// Mitsubishi GX Works2 project: BookEX6_8 Function   PLC: Q13UDV

// global labels: Global
VAR_GLOBAL
  bVar0 AT M5000 : BOOL;
  abArray0 AT M5010 : ARRAY [0..49] OF BOOL;
  sStr0 AT D5000 : STRING[199];
  sStr1 AT D5100 : STRING[199];
  sStr2 AT D5200 : STRING[199];
  sStr3 AT D5300 : STRING[199];
  sStr4 AT D5400 : STRING[199];
  sStr5 AT D5500 : STRING[199];
  sStr6 AT D5600 : STRING[199];
  sStr7 AT D5700 : STRING[199];
  sStr8 AT D5800 : STRING[199];
  sStr9 AT D5900 : STRING[199];
  iVar0 AT D4500 : INT;
  iVar1 AT D4501 : INT;
  iVar2 AT D4502 : INT;
  iVar3 AT D4503 : INT;
  iVar4 AT D4504 : INT;
  iVar5 AT D4505 : INT;
  iVar6 AT D4506 : INT;
  iVar7 AT D4507 : INT;
  iVar8 AT D4508 : INT;
  iVar9 AT D4509 : INT;
  dVar0 AT D4510 : DINT;
  dVar1 AT D4512 : DINT;
  dVar2 AT D4514 : DINT;
  dVar3 AT D4516 : DINT;
  dVar4 AT D4518 : DINT;
  dVar5 AT D4520 : DINT;
  dVar6 AT D4522 : DINT;
  dVar7 AT D4524 : DINT;
  dVar8 AT D4526 : DINT;
  dVar9 AT D4528 : DINT;
  wVar0 AT D4530 : WORD;
  wVar1 AT D4531 : WORD;
  wVar2 AT D4532 : WORD;
  wVar3 AT D4533 : WORD;
  wVar4 AT D4534 : WORD;
  wVar5 AT D4535 : WORD;
  wVar6 AT D4536 : WORD;
  wVar7 AT D4537 : WORD;
  wVar8 AT D4538 : WORD;
  wVar9 AT D4539 : WORD;
  dwVar0 AT D4540 : DWORD;
  dwVar1 AT D4542 : DWORD;
  dwVar2 AT D4544 : DWORD;
  dwVar3 AT D4546 : DWORD;
  dwVar4 AT D4548 : DWORD;
  dwVar5 AT D4550 : DWORD;
  dwVar6 AT D4552 : DWORD;
  dwVar7 AT D4554 : DWORD;
  dwVar8 AT D4556 : DWORD;
  dwVar9 AT D4558 : DWORD;
  fsVar0 AT D4560 : REAL;
  fsVar1 AT D4562 : REAL;
  fsVar2 AT D4564 : REAL;
  fsVar3 AT D4566 : REAL;
  fsVar4 AT D4568 : REAL;
  fsVar5 AT D4570 : REAL;
  fsVar6 AT D4572 : REAL;
  fsVar7 AT D4574 : REAL;
  fsVar8 AT D4576 : REAL;
  fsVar9 AT D4578 : REAL;
  fdVar0 AT D4580 : LREAL;
  tTime0 AT D4620 : TIME;
  tTime1 AT D4622 : TIME;
  tTime2 AT D4624 : TIME;
  tTime3 AT D4626 : TIME;
  tTime4 AT D4628 : TIME;
  tTime5 AT D4630 : TIME;
  tTime6 AT D4632 : TIME;
  tTime7 AT D4634 : TIME;
  tTime8 AT D4636 : TIME;
  tTime9 AT D4638 : TIME;
  tTime10 AT D4640 : TIME;
  bVar1 AT M5001 : BOOL;
  bVar2 AT M5002 : BOOL;
  bVar3 AT M5003 : BOOL;
  bVar4 AT M5004 : BOOL;
  bVar5 AT M5005 : BOOL;
  bVar6 AT M5006 : BOOL;
  bVar7 AT M5007 : BOOL;
  bVar8 AT M5008 : BOOL;
  bVar9 AT M5009 : BOOL;
  abArray1 AT M5060 : ARRAY [0..49] OF BOOL;
  abArray2 AT M5110 : ARRAY [0..49] OF BOOL;
  abArray3 AT M5160 : ARRAY [0..49] OF BOOL;
  abArray4 AT M5210 : ARRAY [0..49] OF BOOL;
  abArray5 AT M5260 : ARRAY [0..49] OF BOOL;
  abArray6 AT M5310 : ARRAY [0..49] OF BOOL;
  abArray7 AT M5360 : ARRAY [0..49] OF BOOL;
  abArray8 AT M5410 : ARRAY [0..49] OF BOOL;
  abArray9 AT M5460 : ARRAY [0..49] OF BOOL;
  fdVar1 AT D4584 : LREAL;
  fdVar2 AT D4588 : LREAL;
  fdVar3 AT D4592 : LREAL;
  fdVar4 AT D4596 : LREAL;
  fdVar5 AT D4600 : LREAL;
  fdVar6 AT D4604 : LREAL;
  fdVar7 AT D4608 : LREAL;
  fdVar8 AT D4612 : LREAL;
  fdVar9 AT D4616 : LREAL;
  afsPen0 AT D2000 : ARRAY [0..499] OF REAL;
  afsPen1 AT D3000 : ARRAY [0..499] OF REAL;
END_VAR
// user libraries (not included): HMI

FUNCTION ACOSH
VAR_INPUT
  fs_IN : REAL;
END_VAR
VAR
  fsTemp1 : REAL;
  fsTemp2 : REAL;
END_VAR
;(* ACOSH *)
ACOSH := LN(fs_IN + SQRT(fs_IN * fs_IN - 1.0));
END_FUNCTION

FUNCTION ASINH
VAR_INPUT
  fs_IN : REAL;
END_VAR
VAR
  fsTemp1 : REAL;
  fsTemp2 : REAL;
END_VAR
;(* ASINH *)
ASINH := LN(fs_IN + SQRT(fs_IN * fs_IN + 1.0));
END_FUNCTION

FUNCTION ATANH
VAR_INPUT
  fs_IN : REAL;
END_VAR
VAR
  fsTemp1 : REAL;
  fsTemp2 : REAL;
END_VAR
;(* ATANH *)
ATANH := LN((1.0 + fs_IN)/(1.0 - fs_IN)) / 2.0;
END_FUNCTION

FUNCTION COSH
VAR_INPUT
  fs_IN : REAL;
END_VAR
VAR
  fsTemp1 : REAL;
  fsTemp2 : REAL;
END_VAR
;(* COSH *)
EXP_E(TRUE, fs_IN, fsTemp1); 
COSH := (1.0 / fsTemp1+fsTemp1) / 2.0;
END_FUNCTION

FUNCTION Day2Time
VAR_INPUT
  fs_IN : REAL;
END_VAR
;
Day2Time := DINT_TO_TIME(REAL_TO_DINT(fs_IN * 86400000.0));
END_FUNCTION

FUNCTION EXP10
VAR_INPUT
  fs_IN : REAL;
END_VAR
VAR
  fsTemp : REAL;
END_VAR
;
EXP_E(TRUE, fs_IN * 2.302585, fsTemp);
EXP10 := fsTemp;
END_FUNCTION

FUNCTION Overlap
VAR_INPUT
  CPos1 : INT;
  CPos2 : INT;
  TPos1 : INT;
  TPos2 : INT;
END_VAR
VAR
  tsPos : INT;
  tePos : INT;
END_VAR
VAR_INPUT
  Safe : INT;
END_VAR
VAR
  tst1 : BOOL;
  tst2 : BOOL;
  tst3 : BOOL;
  tst4 : BOOL;
  csPos : INT;
  cePos : INT;
END_VAR
;
IF TPos1 < TPos2 THEN
	tsPos := TPos1;
	tePos := TPos2;
ELSE
	tsPos := TPos2;
	tePos := TPos1;
END_IF;
IF CPos1 < CPos2 THEN
	csPos := CPos1;
	cePos := CPos2;
ELSE
	csPos := CPos2;
	cePos := CPos1;
END_IF;

tst1 := csPos >= tsPos AND csPos <= tePos;
tst2 := cePos >= tsPos AND cePos <= tePos;
tst3 := ABS(tsPos - cePos) <= Safe;
tst4 := ABS(tePos - csPos) <= Safe;

IF tst1 OR tst2 OR tst3 OR tst4 THEN
	Overlap := TRUE;
ELSE
	Overlap := FALSE;
END_IF;
END_FUNCTION

FUNCTION SINH
VAR_INPUT
  fs_IN : REAL;
END_VAR
VAR
  fsTemp1 : REAL;
  fsTemp2 : REAL;
END_VAR
;(* SINH *)
IF ABS(fs_IN) < 0.002 THEN
	SINH := fs_IN;
ELSE
	EXP_E(TRUE, fs_IN, fsTemp1); 
	EXP_E(TRUE, -fs_IN, fsTemp2); 
	SINH := (fsTemp1 - fsTemp2) / 2.0;
END_IF;
END_FUNCTION

FUNCTION SqrtN
VAR_INPUT
  fs_IN : REAL;
  i_IN : INT;
END_VAR
VAR
  fsTemp : REAL;
END_VAR
;
IF i_IN > 0 THEN
	fsTemp := 1.0 / INT_TO_REAL(i_IN);
	SqrtN := EXPT(fs_IN, fsTemp);
ELSE
	SqrtN := 0.0;
END_IF;
END_FUNCTION

FUNCTION TANH
VAR_INPUT
  fs_IN : REAL;
END_VAR
VAR
  fsTemp1 : REAL;
  fsTemp2 : REAL;
END_VAR
;(* TANH *)
IF fs_IN > 20.0 THEN
	TANH := 1.0;
ELSIF fs_IN < -20.0 THEN
	TANH := -1.0;
ELSE
	EXP_E(TRUE, fs_IN * 2.0, fsTemp1); 
	TANH := 1.0 - 2.0 / (fsTemp1 + 1.0);
END_IF;
END_FUNCTION

PROGRAM ExABS
(* structured ladder/FBD written out as ST: instructions are called as NAME(EN, inputs, outputs); _pN, _eN, _tN stand for wires *)
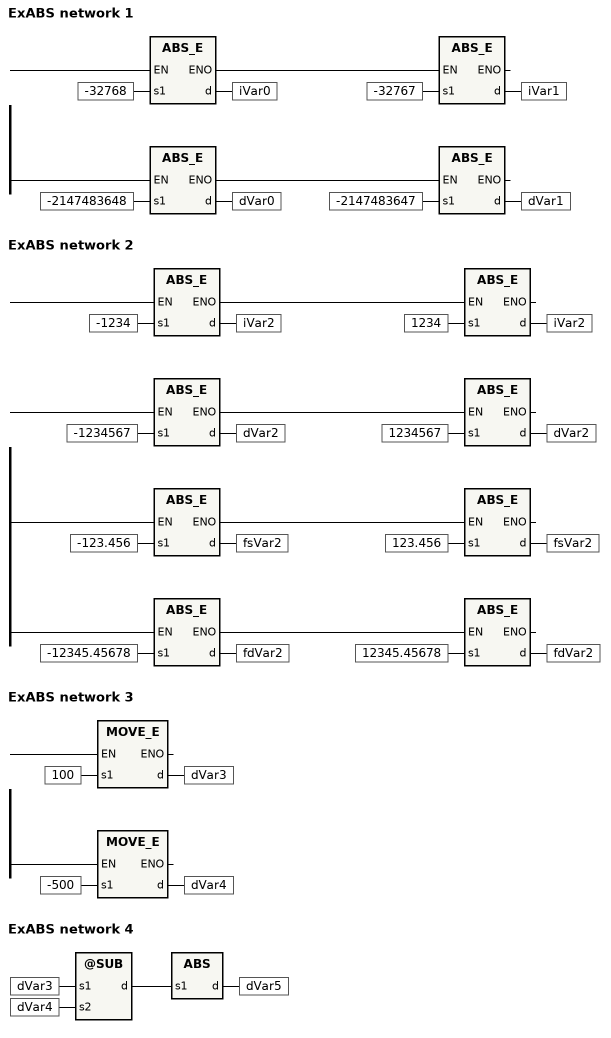
(* network 1 *)
_e1 := ABS_E(TRUE, -32768, iVar0);
ABS_E(_e1, -32767, iVar1);
_e2 := ABS_E(TRUE, -2147483648, dVar0);
ABS_E(_e2, -2147483647, dVar1);
(* network 2 *)
_e1 := ABS_E(TRUE, -1234, iVar2);
ABS_E(_e1, 1234, iVar2);
_e2 := ABS_E(TRUE, -1234567, dVar2);
ABS_E(_e2, 1234567, dVar2);
_e3 := ABS_E(TRUE, -123.456, fsVar2);
ABS_E(_e3, 123.456, fsVar2);
_e4 := ABS_E(TRUE, -12345.45678, fdVar2);
ABS_E(_e4, 12345.45678, fdVar2);
(* network 3 *)
MOVE_E(TRUE, 100, dVar3);
MOVE_E(TRUE, -500, dVar4);
(* network 4 *)
dVar5 := ABS(@SUB(dVar3, dVar4));
END_PROGRAM

PROGRAM ExASinGraph
VAR
  ix : INT;
  radx : REAL;
  fsx1 : REAL;
  fsx2 : REAL;
  fscale : REAL;
END_VAR
 
IF SM402 THEN
	fsVar0 := 0.0;		(* Offset X *)
	fsVar1 := 0.0;		(* Offset Y *)
	fsVar2 := 1.0;		(* Radius X *)
	fsVar3 := 1.0;		(* Radius Y *)
	fsVar4 := 1.0;		(* Scale X *)
	fsVar5 := 1.0;		(* Scale Y *)
	iVar0 := 0;				(* Type *)
	iVar1 := 0;				(* Count *)
END_IF;

CASE iVar0 OF 
 	13 : (* ASIN *)
		fsVar6 := -1.0;		 (* MIN X *)
		fsVar7 := 1.0; 		 (* MAX X *)	
		fsVar8 := -2.0;		 (* MIN Y *)
		fsVar9 := 2.0;		 (* MAX Y *)	
		FOR ix := 0 TO 359 DO
			fscale := fsVar7 * 2.0 * INT_TO_REAL(ix) / 360.0;
			afsPen0[ix] := (fscale - fsVar7) * fsVar4;
			ASIN_E(TRUE, afsPen0[ix] , fsx2);
			afsPen1[ix] := fsx2 * fsVar5;
		END_FOR;  
 	14 : (* ACOS *)
		fsVar6 := -1.0;		 (* MIN X *)
		fsVar7 := 1.0; 		 (* MAX X *)	
		fsVar8 := -3.5;		 (* MIN Y *)
		fsVar9 := 3.5;		 (* MAX Y *)	
		FOR ix := 0 TO 359 DO
			fscale := fsVar7 * 2.0 * INT_TO_REAL(ix) / 360.0;
			afsPen0[ix] := (fscale - fsVar7) * fsVar4;
			ACOS_E(TRUE, afsPen0[ix], fsx2);
			afsPen1[ix] := fsx2 * fsVar5;
		END_FOR;  
 	15 : (* ATAN *)
		fsVar6 := -12.0;		 (* MIN X *)
		fsVar7 := 12.0; 		 (* MAX X *)	
		fsVar8 := -2.0;		 (* MIN Y *)
		fsVar9 := 2.0;		 (* MAX Y *)	
		FOR ix := 0 TO 359 DO
			fscale := fsVar7 * 2.0 * INT_TO_REAL(ix) / 360.0;
			afsPen0[ix] := (fscale - fsVar7) * fsVar4;
			ATAN_E(TRUE, afsPen0[ix], fsx2);
			afsPen1[ix] := fsx2 * fsVar5;
		END_FOR;  
END_CASE;
END_PROGRAM

PROGRAM ExASinhGraph
VAR
  ix : INT;
  radx : REAL;
  fsx1 : REAL;
  fsx2 : REAL;
  fscale : REAL;
END_VAR
 
IF SM402 THEN
	fsVar0 := 0.0;		(* Offset X *)
	fsVar1 := 0.0;		(* Offset Y *)
	fsVar2 := 1.0;		(* Radius X *)
	fsVar3 := 1.0;		(* Radius Y *)
	fsVar4 := 1.0;		(* Scale X *)
	fsVar5 := 1.0;		(* Scale Y *)
	iVar0 := 0;				(* Type *)
	iVar1 := 0;				(* Count *)
END_IF;

CASE iVar0 OF 
 	1 : (* ASINH *)
		fsVar6 := -12.0;		 (* MIN X *)
		fsVar7 := 12.0; 		 (* MAX X *)	
		fsVar8 := -6.0;		 (* MIN Y *)
		fsVar9 := 6.0;		 (* MAX Y *)	
		FOR ix := 0 TO 359 DO
			fscale := fsVar7 * 2.0 * INT_TO_REAL(ix) / 360.0;
			afsPen0[ix] := (fscale - fsVar7) * fsVar4;
			fsx2 := ASINH(afsPen0[ix]);
			afsPen1[ix] := fsx2 * fsVar5;
		END_FOR;  
 	2 : (* ACOSH *)
		fsVar6 := -12.0;		 (* MIN X *)
		fsVar7 := 12.0; 		 (* MAX X *)	
		fsVar8 := -6.0;		 (* MIN Y *)
		fsVar9 := 6.0;		 (* MAX Y *)	
		FOR ix := 0 TO 359 DO
			fscale := fsVar7 * 2.0 * INT_TO_REAL(ix) / 360.0;
			IF (fscale - fsVar7) * fsVar4 < 1.0 THEN
				afsPen0[ix] := 0.0;
				afsPen1[ix] := 0.0;
			ELSE
				afsPen0[ix] := (fscale - fsVar7) * fsVar4;
				fsx2 := ACOSH(afsPen0[ix]);
				afsPen1[ix] := fsx2 * fsVar5;
			END_IF;
		END_FOR;  
 	3 : (* ATANH *)
		fsVar6 := -0.9;		 (* MIN X *)
		fsVar7 := 0.9; 		 (* MAX X *)	
		fsVar8 := -2.0;		 (* MIN Y *)
		fsVar9 := 2.0;		 (* MAX Y *)	
		FOR ix := 0 TO 359 DO
			fscale := fsVar7 * 2.0 * INT_TO_REAL(ix) / 360.0;
			afsPen0[ix] := (fscale - fsVar7) * fsVar4;
			fsx2 := ATANH(afsPen0[ix]);
			afsPen1[ix] := fsx2 * fsVar5;
		END_FOR;  
END_CASE;
END_PROGRAM

PROGRAM ExCircle
VAR
  ix : INT;
  radx : REAL;
  fsx1 : REAL;
  fsx2 : REAL;
  fscale : REAL;
END_VAR
 
IF SM402 THEN
	fsVar0 := 0.0;		(* Offset X *)
	fsVar1 := 0.0;		(* Offset Y *)
	fsVar2 := 1.0;		(* Radius X *)
	fsVar3 := 1.0;		(* Radius Y *)
	fsVar4 := 1.0;		(* Scale X *)
	fsVar5 := 1.0;		(* Scale Y *)
	fsVar6 := -1.0;		(* MIN X *)
	fsVar7 := 1.0; 		(* MAX X *)	
	fsVar8 := -1.0;		(* MIN Y *)
	fsVar9 := 1.0;		(* MAX Y *)	
	iVar0 := 0;				(* Type *)
	iVar1 := 0;				(* Count *)
END_IF;

CASE iVar0 OF 
	0 : (* Circle *)
		FOR ix := 0 TO 359 DO
			RAD(TRUE,INT_TO_REAL(ix),radx);
			COS(TRUE, radx, fsx1);
			afsPen0[ix] := fsx1 * fsVar2 * fsVar4 + fsVar0;
			SIN(TRUE, radx, fsx2);
			afsPen1[ix] := fsx2 * fsVar3 * fsVar5 + fsVar1;
		END_FOR;
		iVar1 := 0;
	1 : (* Slow Circle *)
		CASE iVar1 OF
			0 :
				FOR ix := 0 TO 359 DO
					afsPen0[ix] := 0.0;
					afsPen1[ix] := 0.0;;
				END_FOR;
				iVar1 := 1;
			1..360 :
				RAD(TRUE,INT_TO_REAL(iVar1-1),radx);
				COS(TRUE, radx, fsx1);
				afsPen0[iVar1-1] := fsx1 * fsVar2 * fsVar4 + fsVar0;
				SIN(TRUE, radx, fsx2);
				afsPen1[iVar1-1] := fsx2 * fsVar3 * fsVar5 + fsVar1;
				iVar1 := iVar1 + 1;
			ELSE
				iVar1 := 0;
		END_CASE;
END_CASE;
END_PROGRAM

PROGRAM ExEXP10
(* structured ladder/FBD written out as ST: instructions are called as NAME(EN, inputs, outputs); _pN, _eN, _tN stand for wires *)
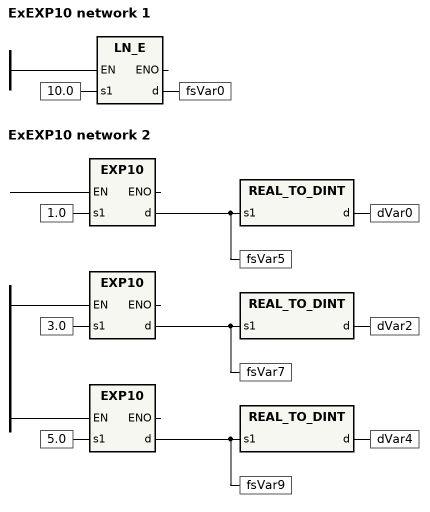
(* network 1 *)
LN_E(TRUE, 10.0, fsVar0);
(* network 2 *)
EXP10(TRUE, 1.0, fsVar5);
dVar0 := REAL_TO_DINT(fsVar5);
EXP10(TRUE, 3.0, fsVar7);
dVar2 := REAL_TO_DINT(fsVar7);
EXP10(TRUE, 5.0, fsVar9);
dVar4 := REAL_TO_DINT(fsVar9);
END_PROGRAM

PROGRAM ExLnEXP
(* structured ladder/FBD written out as ST: instructions are called as NAME(EN, inputs, outputs); _pN, _eN, _tN stand for wires *)
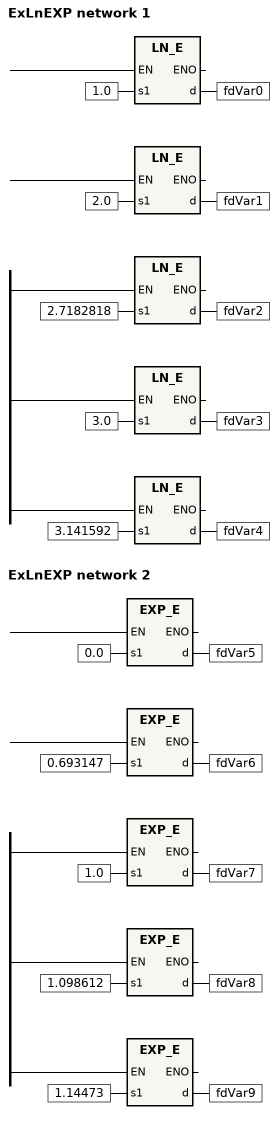
(* network 1 *)
LN_E(TRUE, 1.0, fdVar0);
LN_E(TRUE, 2.0, fdVar1);
LN_E(TRUE, 2.7182818, fdVar2);
LN_E(TRUE, 3.0, fdVar3);
LN_E(TRUE, 3.141592, fdVar4);
(* network 2 *)
EXP_E(TRUE, 0.0, fdVar5);
EXP_E(TRUE, 0.693147, fdVar6);
EXP_E(TRUE, 1.0, fdVar7);
EXP_E(TRUE, 1.098612, fdVar8);
EXP_E(TRUE, 1.14473, fdVar9);
END_PROGRAM

PROGRAM ExLnGraph
VAR
  ix : INT;
  radx : REAL;
  fsx1 : REAL;
  fsx2 : REAL;
  fscale : REAL;
END_VAR
 
IF SM402 THEN
	fsVar0 := 0.0;		(* Offset X *)
	fsVar1 := 0.0;		(* Offset Y *)
	fsVar2 := 1.0;		(* Radius X *)
	fsVar3 := 1.0;		(* Radius Y *)
	fsVar4 := 1.0;		(* Scale X *)
	fsVar5 := 1.0;		(* Scale Y *)
	iVar0 := 0;				(* Type *)
	iVar1 := 0;				(* Count *)
	FOR ix := 0 TO 359 DO
		afsPen0[ix] := 0.0;
		afsPen1[ix] := 0.0;;
	END_FOR;
END_IF;
	
CASE iVar0 OF 
	0 : (* Ln *)
		fsVar6 := -12.0;		(* MIN X *)
		fsVar7 := 12.0; 		(* MAX X *)	
		fsVar8 := -6.0;		(* MIN Y *)
		fsVar9 := 6.0;		(* MAX Y *)	
		FOR ix := 1 TO 180 DO
			fsx1 := fsVar7 * INT_TO_REAL(ix) / 180.0;
			LN_E( TRUE, fsx1, fsx2); 
			afsPen0[ix] := fsx1;
			afsPen1[ix] := fsx2;
		END_FOR;
		iVar1 := 0;
	1 : (* Log10 *)
		fsVar6 := -4.0;		(* MIN X *)
		fsVar7 := 4.0; 		(* MAX X *)	
		fsVar8 := -4.0;		(* MIN Y *)
		fsVar9 := 4.0;		(* MAX Y *)	
		FOR ix := 0 TO 359 DO
			fsx1 := fsVar7 * 2.0 * INT_TO_REAL(ix - 180) / 360.0;
			EXP_E(TRUE, fsx1, fsx2); 
			afsPen0[ix] := fsx1;
			afsPen1[ix] := fsx2;
		END_FOR;
		iVar1 := 0;
END_CASE;
END_PROGRAM

PROGRAM ExOverlap
(* structured ladder/FBD written out as ST: instructions are called as NAME(EN, inputs, outputs); _pN, _eN, _tN stand for wires *)
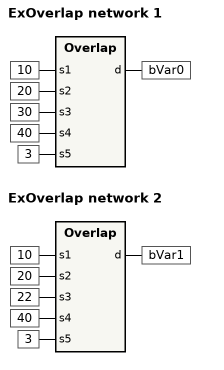
(* network 1 *)
bVar0 := Overlap(10, 20, 30, 40, 3);
(* network 2 *)
bVar1 := Overlap(10, 20, 22, 40, 3);
END_PROGRAM

PROGRAM ExSinGraph
VAR
  ix : INT;
  radx : REAL;
  fsx1 : REAL;
  fsx2 : REAL;
  fscale : REAL;
END_VAR
 
IF SM402 THEN
	fsVar0 := 0.0;		(* Offset X *)
	fsVar1 := 0.0;		(* Offset Y *)
	fsVar2 := 1.0;		(* Radius X *)
	fsVar3 := 1.0;		(* Radius Y *)
	fsVar4 := 1.0;		(* Scale X *)
	fsVar5 := 1.0;		(* Scale Y *)
	fsVar6 := -1.0;		 (* MIN X *)
	fsVar7 := 1.0; 		 (* MAX X *)	
	fsVar8 := -1.0;		 (* MIN Y *)
	fsVar9 := 1.0;		 (* MAX Y *)	
	iVar0 := 0;				(* Type *)
	iVar1 := 0;				(* Count *)
END_IF;

CASE iVar0 OF 
	10 : (* SIN *)
		FOR ix := 0 TO 359 DO
			RAD(TRUE,INT_TO_REAL(ix),radx);
			SIN_E(TRUE, radx, fsx2);
			fscale := fsVar7 * 2.0 * INT_TO_REAL(ix)  / 360.0;
			afsPen0[ix] := (fscale - fsVar7) * fsVar4;
			afsPen1[ix] := fsx2 * fsVar5;
		END_FOR;  
 	11 : (* COS *)
		FOR ix := 0 TO 359 DO
			RAD(TRUE,INT_TO_REAL(ix),radx);
			COS_E(TRUE, radx, fsx2);
			fscale := fsVar7 * 2.0 * INT_TO_REAL(ix) / 360.0;
			afsPen0[ix] := (fscale - fsVar7) * fsVar4;
			afsPen1[ix] := fsx2 * fsVar5;
		END_FOR;  
 	12 : (* TAN *)
		FOR ix := 0 TO 359 DO
			RAD(TRUE,INT_TO_REAL(ix),radx);
			TAN_E(TRUE, radx, fsx2);
			fscale := fsVar7 * 2.0 * INT_TO_REAL(ix) / 360.0;
			afsPen0[ix] := (fscale - fsVar7) * fsVar4;
			afsPen1[ix] := fsx2 * fsVar5;
		END_FOR;  
END_CASE;
END_PROGRAM

PROGRAM ExSinhGraph
VAR
  ix : INT;
  radx : REAL;
  fsx1 : REAL;
  fsx2 : REAL;
  fscale : REAL;
END_VAR
 
IF SM402 THEN
	fsVar0 := 0.0;		(* Offset X *)
	fsVar1 := 0.0;		(* Offset Y *)
	fsVar2 := 1.0;		(* Radius X *)
	fsVar3 := 1.0;		(* Radius Y *)
	fsVar4 := 1.0;		(* Scale X *)
	fsVar5 := 1.0;		(* Scale Y *)
	iVar0 := 0;				(* Type *)
	iVar1 := 0;				(* Count *)
END_IF;

CASE iVar0 OF 
 	1 : (* SINH *)
		fsVar6 := -2.5;		 (* MIN X *)
		fsVar7 := 2.5; 		 (* MAX X *)	
		fsVar8 := -6.0;		 (* MIN Y *)
		fsVar9 := 6.0;		 (* MAX Y *)	
		FOR ix := 0 TO 359 DO
			fscale := fsVar7 * 2.0 * INT_TO_REAL(ix) / 360.0;
			afsPen0[ix] := (fscale - fsVar7) * fsVar4;
			fsx2 := SINH(afsPen0[ix]);
			afsPen1[ix] := fsx2 * fsVar5;
		END_FOR;  
 	2 : (* COSH *)
		fsVar6 := -3.4;		 (* MIN X *)
		fsVar7 := 3.4; 		 (* MAX X *)	
		fsVar8 := -15.0;		 (* MIN Y *)
		fsVar9 := 15.0;		 (* MAX Y *)	
		FOR ix := 0 TO 359 DO
			fscale := fsVar7 * 2.0 * INT_TO_REAL(ix) / 360.0;
			afsPen0[ix] := (fscale - fsVar7) * fsVar4;
			fsx2 := COSH(afsPen0[ix]);
			afsPen1[ix] := fsx2 * fsVar5;
		END_FOR;  
 	3 : (* TANH *)
		fsVar6 := -6.0;		 (* MIN X *)
		fsVar7 := 6.0; 		 (* MAX X *)	
		fsVar8 := -2.0;		 (* MIN Y *)
		fsVar9 := 2.0;		 (* MAX Y *)	
		FOR ix := 0 TO 359 DO
			fscale := fsVar7 * 2.0 * INT_TO_REAL(ix) / 360.0;
			afsPen0[ix] := (fscale - fsVar7) * fsVar4;
			fsx2 := TANH(afsPen0[ix]);
			afsPen1[ix] := fsx2 * fsVar5;
		END_FOR;  
END_CASE;
END_PROGRAM

PROGRAM ExSQRT
(* structured ladder/FBD written out as ST: instructions are called as NAME(EN, inputs, outputs); _pN, _eN, _tN stand for wires *)
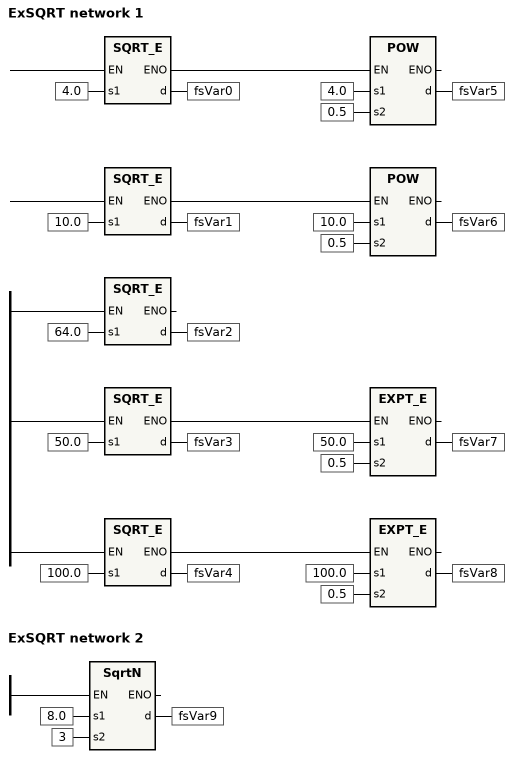
(* network 1 *)
_e1 := SQRT_E(TRUE, 4.0, fsVar0);
POW(_e1, 4.0, 0.5, fsVar5);
_e2 := SQRT_E(TRUE, 10.0, fsVar1);
POW(_e2, 10.0, 0.5, fsVar6);
SQRT_E(TRUE, 64.0, fsVar2);
_e3 := SQRT_E(TRUE, 50.0, fsVar3);
EXPT_E(_e3, 50.0, 0.5, fsVar7);
_e4 := SQRT_E(TRUE, 100.0, fsVar4);
EXPT_E(_e4, 100.0, 0.5, fsVar8);
(* network 2 *)
SqrtN(TRUE, 8.0, 3, fsVar9);
END_PROGRAM

FUNCTION ATAN2
VAR_INPUT
  PosX : LREAL;
  PosY : LREAL;
END_VAR
VAR CONSTANT
  fdPI : LREAL := 3.14159265;
END_VAR
VAR
  fdRad : LREAL;
END_VAR
;

IF PosX > 0.0 THEN													
    ATAN_E(TRUE, PosY / PosX, fdRad);
ELSIF (PosX < 0.0) AND (PosY >= 0.0) THEN	
    ATAN_E(TRUE, PosY / PosX, fdRad); 
    fdRad := fdRad + fdPI;
ELSIF (PosX < 0.0) AND (PosY < 0.0) THEN	
    ATAN_E(TRUE, PosY / PosX, fdRad); 
    fdRad := fdRad - fdPI;
ELSIF (PosX = 0.0) AND (PosY > 0.0) THEN	
    fdRad := fdPI/ 2.0;
ELSIF (PosX = 0.0) AND (PosY < 0.0) THEN		
    fdRad := - (fdPI/ 2.0);
ELSE																					
    fdRad := 0.0;
END_IF;

ATAN2 := fdRad * (180.0 / fdPI);
END_FUNCTION

PROGRAM ExATAN2
(* structured ladder/FBD written out as ST: instructions are called as NAME(EN, inputs, outputs); _pN, _eN, _tN stand for wires *)
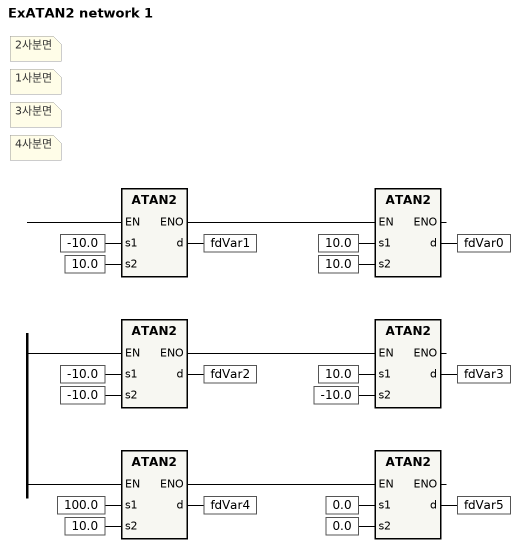
(* network 1 *)
(* 2사분면 *)
(* 1사분면 *)
(* 3사분면 *)
(* 4사분면 *)
_e1 := ATAN2(TRUE, -10.0, 10.0, fdVar1);
ATAN2(_e1, 10.0, 10.0, fdVar0);
_e2 := ATAN2(TRUE, -10.0, -10.0, fdVar2);
ATAN2(_e2, 10.0, -10.0, fdVar3);
_e3 := ATAN2(TRUE, 100.0, 10.0, fdVar4);
ATAN2(_e3, 0.0, 0.0, fdVar5);
END_PROGRAM

PROGRAM ExTemp
(* structured ladder/FBD written out as ST: instructions are called as NAME(EN, inputs, outputs); _pN, _eN, _tN stand for wires *)
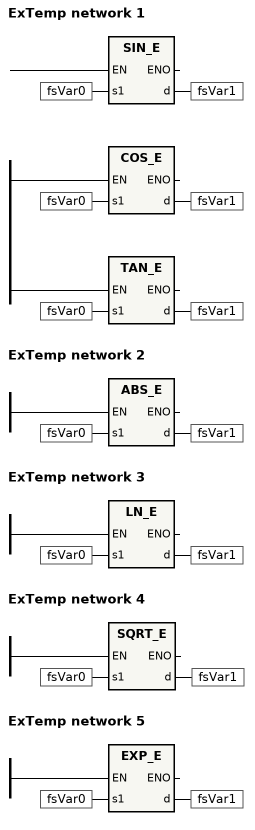
(* network 1 *)
SIN_E(TRUE, fsVar0, fsVar1);
COS_E(TRUE, fsVar0, fsVar1);
TAN_E(TRUE, fsVar0, fsVar1);
(* network 2 *)
ABS_E(TRUE, fsVar0, fsVar1);
(* network 3 *)
LN_E(TRUE, fsVar0, fsVar1);
(* network 4 *)
SQRT_E(TRUE, fsVar0, fsVar1);
(* network 5 *)
EXP_E(TRUE, fsVar0, fsVar1);
END_PROGRAM

PROGRAM ExExpGraph
VAR
  ix : INT;
  radx : REAL;
  fsx1 : REAL;
  fsx2 : REAL;
  fscale : REAL;
  fsTemp : REAL;
  fsExp : REAL;
  fsx3 : REAL;
  iy : INT;
END_VAR
 
fsVar8 := 1.0;
fsVar9 := -1.0;

FOR ix := 0 TO 359 DO
	iy := ix-180;
	fsTemp := INT_TO_REAL(iy); 
	fsTemp := fsTemp / 36.0;
	 
	EXP_E(TRUE, fsTemp * 2.0, fsExp);
	fsx3 := fsExp;
	fsx1 := fsExp + 1.0;
	fsx2 := fsx3 / fsx1;
	afsPen0[ix] := fsx2;
	
	EXP_E(TRUE, -fsTemp, fsExp);
	fsx3 := 1.0;
	fsx1 := fsExp + 1.0;
	fsx2 := fsx3 / fsx1;
	afsPen1[ix] := fsx2; 
END_FOR;
END_PROGRAM

PROGRAM ExGetWave
VAR
  GenWave_1 : GenWave;
  GenWave_2 : GenWave;
  GenWave_3 : GenWave;
  GenWave_4 : GenWave;
END_VAR
(* structured ladder/FBD written out as ST: instructions are called as NAME(EN, inputs, outputs); _pN, _eN, _tN stand for wires *)
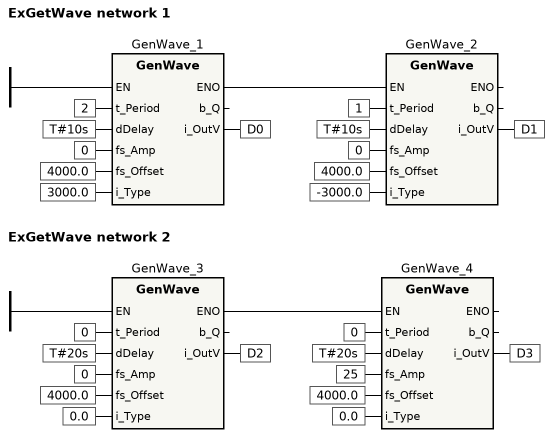
(* network 1 *)
GenWave_1(EN := TRUE, t_Period := 2, dDelay := T#10s, fs_Amp := 0, fs_Offset := 4000.0, i_Type := 3000.0, i_OutV => D0);
GenWave_2(EN := GenWave_1.ENO, t_Period := 1, dDelay := T#10s, fs_Amp := 0, fs_Offset := 4000.0, i_Type := -3000.0, i_OutV => D1);
(* network 2 *)
GenWave_3(EN := TRUE, t_Period := 0, dDelay := T#20s, fs_Amp := 0, fs_Offset := 4000.0, i_Type := 0.0, i_OutV => D2);
GenWave_4(EN := GenWave_3.ENO, t_Period := 0, dDelay := T#20s, fs_Amp := 25, fs_Offset := 4000.0, i_Type := 0.0, i_OutV => D3);
END_PROGRAM

FUNCTION_BLOCK GenWave
VAR_INPUT
  t_Period : TIME;
  dDelay : DINT;  (* % *)
  fs_Amp : REAL;
  fs_Offset : REAL;
END_VAR
VAR_OUTPUT
  b_Q : BOOL;
  i_OutV : INT;
END_VAR
VAR
  fsTemp : REAL;
  fsTemp1 : REAL;
  tLast : TIME;
  tPast : TIME;
  tCurr : TIME;
  tMulTime : TIME;
  tShift : TIME;
  dSftTime : DINT;
  bInit : BOOL;
  qTemp : BOOL;
END_VAR
VAR CONSTANT
  PI2 : REAL := 6.283185;
END_VAR
VAR
  fbTON : TON;
END_VAR
VAR_INPUT
  i_Type : INT;
END_VAR
VAR
  dMulTime : DINT;
  dHalfPeriod : DINT;
END_VAR
;
fbTON(IN := NOT qTemp, PT := T#30m, Q:= qTemp, ET := tPast);
tCurr := tPast - tLast;

IF NOT bInit THEN
	bInit := TRUE;
	tLast := tCurr;
	tCurr := T#0s;
END_IF;

IF tCurr >= t_Period THEN
	tLast := tLast + t_Period;
	tCurr := tCurr - t_Period;
END_IF;

CASE i_Type OF 
	0 : (* SIN *)
		IF t_Period > T#0s THEN
			dSftTime := TIME_TO_DINT(t_Period) * dDelay / 100;
			tShift := DINT_TO_TIME(dSftTime);
			tMulTime := tCurr - tShift;
			fsTemp1 := PI2 * DINT_TO_REAL(TIME_TO_DINT(tMulTime)) / DINT_TO_REAL(TIME_TO_DINT(t_Period));
			SIN(TRUE, fsTemp1, fsTemp);
		ELSE
			fsTemp := 0.0;
		END_IF;
	1 : (* SQUARE *)
		IF t_Period > T#0s THEN
			dMulTime := TIME_TO_DINT(tCurr);
			dHalfPeriod := TIME_TO_DINT(t_Period) / 2;
			IF dMulTime < dHalfPeriod THEN
				fsTemp := 1.0;
			ELSE
				fsTemp := -1.0;
			END_IF;
		ELSE
			fsTemp := 0.0;
		END_IF; 
	2 : (* SAW *)
		IF t_Period > T#0s THEN
			fsTemp := DINT_TO_REAL(TIME_TO_DINT(tCurr) * 2) / DINT_TO_REAL(TIME_TO_DINT(t_Period)) - 1.0;
		ELSE
			fsTemp := 0.0;
		END_IF;
END_CASE;
i_OutV := REAL_TO_INT(fs_Amp * fsTemp * 0.5  + fs_Offset);
b_Q := i_OutV < 0;
END_FUNCTION_BLOCK
